{attribute 'qualified_only'}
{attribute 'strict'}
TYPE eTcoEq2TransferConfiguration :
(
	SingleInDoubleOut := 1,
	DoubleInSingleOut := 2,
	SingleInDoubleOutNoPrestopper := 3

);
END_TYPE

(* stored: Version 1.1.0.1
   DUT eTcoEq2TransferConfiguration: Id {da3a245f-571a-4125-8644-d8ce75afb788} *)
